Universal Robots PolyScope program: test_circ_motion4.urp

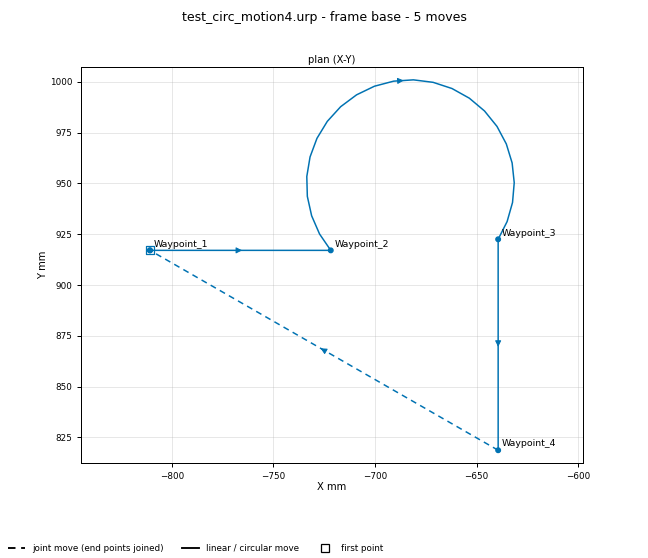
[picture p0: tool path of test_circ_motion4.urp in frame base, 5 of 6 moves have a stored position in this frame; points joined in program order, loops and branches not executed]
Program test_circ_motion4 (installation=default directory=/programs createdIn=5.14.5 lastSavedIn=5.14.5 robotSerialNumber=20236801216)
Calibrated DH parameters: a=[-0.000021, -0.748897, -0.28186, -0.00004, -0.000055, 0]; d=[0.236225, -424.082933, -1564.66872, 1988.95162, 0.159094, 0.153873]; alpha=[1.570844, 0.001002, 0.000337, 1.571488, -1.569996, 0]; deltaTheta=[0, -0.516316, 5.626292, 1.173211, 0.000001, 0]
InitVariablesNode
Robot Program (runOnlyOnce=false)
  MoveP speed 20 mm/s, acceleration 1200 mm/s^2 (blendRadius=0.025 useActiveTCP=true) feature=Base
    Waypoint Waypoint_1: TCP in base x=-810.734 y=917.065 z=-8.085 mm, rx=1.5708 ry=0 rz=0 rad; joints [-61.768, -25.564, 64.413, -38.748, -61.825, -0.129] deg; TCP offset x=0 y=0 z=19 mm, rx=0 ry=0 rz=0 rad
    Waypoint Waypoint_2: TCP in base x=-721.778 y=917.058 z=-8.079 mm, rx=1.5708 ry=0 rz=0 rad; joints [-65.23, -28.38, 71.151, -42.68, -65.286, -0.12] deg
    CircleMove (OrientationMode=FIXED)
      Waypoint ViaPoint_1: TCP in base x=-639.229 y=922.81 z=-11.188 mm, rx=1.501 ry=-0.563 rz=-0.6403 rad; joints [-73.421, -34.524, 86.946, -51.705, -29.477, -3.545] deg
      Waypoint Waypoint_3: TCP in base x=-639.42 y=922.506 z=-11.178 mm, rx=1.2117 ry=-1.2775 rz=-1.3164 rad; joints [-73.921, -40.137, 101.724, -59.15, 22.141, -5.297] deg
    Waypoint Waypoint_4: TCP in base x=-639.414 y=818.709 z=-11.176 mm, rx=1.2117 ry=-1.2775 rz=-1.3165 rad; joints [-72.1, -42.926, 110.242, -65.046, 23.962, -5.112] deg
  MoveJ speed 60 deg/s, acceleration 80 deg/s^2 (useActiveTCP=true) feature=Base
    Waypoint Waypoint_1: TCP in base x=-810.734 y=917.065 z=-8.085 mm, rx=1.5708 ry=0 rz=0 rad; joints [-61.768, -25.564, 64.413, -38.748, -61.825, -0.129] deg
